{attribute 'enable_dynamic_creation'}
FUNCTION_BLOCK FB_Septum EXTENDS FB_UsingPiece
VAR_INPUT
END_VAR
VAR_OUTPUT
END_VAR
VAR
	pVial : POINTER TO FB_Vial;
END_VAR

METHOD FB_init : BOOL
VAR_INPUT
	bInitRetains : BOOL; // if TRUE, the retain variables are initialized (warm start / cold start)
	bInCopyCode : BOOL;  // if TRUE, the instance afterwards gets moved into the copy code (online change)
END_VAR
bUsingPiece := TRUE;
eObjectType := E_ObjectType.OBJECTTYPE_Septum;
eObjectGroup := E_ObjectGroup.OBJECTGROUP_Piece;
END_METHOD

{attribute 'object_name' := 'M_ClearAllProps'}
METHOD M_ClearAllProps

VAR_INPUT
	bIgnoreParent : BOOL; //Es wird das gesamte OD gelöscht. -> Zeiger auf Parent nicht mehr gültig!
END_VAR
pVial := 0;
SUPER^.M_ClearAllProps(bIgnoreParent);
END_METHOD

PROPERTY P_pVial : POINTER TO FB_PieceBase
GET
P_pVial := pVial;
END_GET
SET
pVial := P_pVial;
END_SET
END_PROPERTY

END_FUNCTION_BLOCK

(* stored: Version 1.1.0.1, ProductVersion 3.1.4022.18
   POU FB_Septum: Id {6f242a65-012c-401f-acec-1fd4f959004c}, SpecialFunc None
   Method FB_init: Id {c0096feb-b959-49c1-a46d-713ee6189f09}
   Method M_ClearAllProps: Id {a660089d-e3a0-412f-9f4e-be7015d93b6d}
   Property P_pVial: Id {44ce96bd-185a-4404-b4d6-3d922b850546}
   Get Get: Id {1e6be827-27d5-43b3-8692-4690dd2f75f5}
   Set Set: Id {2034211f-765f-41d6-910e-09588b416d1f} *)
